                $ 887 "A_Touch_p[A_sel_v]=touch_xyz_get_middle(vr2_p1,vr2_p2,vr2_p3,vr2_p4)"
                A_Touch_p[A_sel_v]=touch_xyz_get_middle(vr2_p1,vr2_p2,vr2_p3,vr2_p4)
                $ 888 "var_4≔A_Touch_p[A_sel_v]"
                global var_4=A_Touch_p[A_sel_v]
                $ 889 "var_4≔pose_trans(var_4, p[a6_callar_vert/1000,0,0,0,0,0])"
                global var_4= pose_trans (var_4, p[a6_callar_vert/1000,0,0,0,0,0])
                $ 890 "var_5≔get_actual_tcp_pose()"
                global var_5= get_actual_tcp_pose ()
                $ 891 "var_5[2]=var_4[2]"
                var_5[2]=var_4[2]
                $ 892 "var_5≔pose_trans(var_5, p[0,0,0,0,d2r(10),0])"
                global var_5= pose_trans (var_5, p[0,0,0,0,d2r(10),0])
                $ 893 "MoveL"
                $ 894 "var_5" "breakAfter"
                movel(pose_trans(Base, var_5), a=0.1, v=0.1)
                $ 895 "vr2_p1_up≔contact_fun(p[0,0,0,0,0,0],[1,0,0],20000,20,20)"
                global vr2_p1_up=contact_fun(p[0,0,0,0,0,0],[1,0,0],20000,20,20)
                $ 896 "direction(p[0,0,0,0,0,0],[-1,0,0],20,120,160)"
                direction(p[0,0,0,0,0,0],[-1,0,0],20,120,160)
                $ 897 "direction(p[0,0,0,0,0,0],[0,1,0],10,120,160)"
                direction(p[0,0,0,0,0,0],[0,1,0],10,120,160)
                $ 898 "vr2_p2_up≔contact_fun(p[0,0,0,0,0,0],[1,0,0],20000,20,20)"
                global vr2_p2_up=contact_fun(p[0,0,0,0,0,0],[1,0,0],20000,20,20)
                $ 899 "direction(p[0,0,0,0,0,0],[-1,0,0],14,120,160)"
                direction(p[0,0,0,0,0,0],[-1,0,0],14,120,160)
                $ 900 "vr2_p3_up≔contact_fun(p[0,0,0,0,0,0],[0,1,0],20000,20,20)"
                global vr2_p3_up=contact_fun(p[0,0,0,0,0,0],[0,1,0],20000,20,20)
                $ 901 "direction(p[0,0,0,0,0,0],[0,-1,0],30,120,160)"
                direction(p[0,0,0,0,0,0],[0,-1,0],30,120,160)
                $ 902 "direction(p[0,0,0,0,0,0],[-1,0,0],20,120,160)"
                direction(p[0,0,0,0,0,0],[-1,0,0],20,120,160)
              end
              $ 903 "A_Touch_p[A_sel_v+9]=touch_4point(vr2_p1_up,vr2_p2_up,vr2_p3_up)"
              A_Touch_p[A_sel_v+9]=touch_4point(vr2_p1_up,vr2_p2_up,vr2_p3_up)
              $ 904 "A_Touch_p[A_sel_v+9]=ori_pose(A_Touch_p[A_sel_v+9],A_Touch_p[A_sel_v])"
              A_Touch_p[A_sel_v+9]=ori_pose(A_Touch_p[A_sel_v+9],A_Touch_p[A_sel_v])
            else:
              $ 905 "Else" "noBreak"
              $ 906 "If A_Touch_p[A_VR1]≟p[0,0,0,0,0,0]"
              if (A_Touch_p[A_VR1] == p[0,0,0,0,0,0]):
                $ 907 "Call MoveandTouchFun_3f"
                MoveandTouchFun_3f()
                $ 908 "touch_tmp≔A_Touch_p[A_sel_v]"
                global touch_tmp=A_Touch_p[A_sel_v]
                $ 909 "If A_Prepos_l[A_HOR_MR]≟p[0,0,0,0,0,0]"
                if (A_Prepos_l[A_HOR_MR] == p[0,0,0,0,0,0]):
                  $ 910 "direction(p[0,0,0,0,0,0],[0,1,0],8,120,160)"
                  direction(p[0,0,0,0,0,0],[0,1,0],8,120,160)
                  $ 911 "AAgcp≔get_actual_tcp_pose()"
                  global AAgcp= get_actual_tcp_pose ()
                  $ 912 "AAgangle≔up_right"
                  global AAgangle=p[.445203173045, -.406687378356, -.031125942276, 2.308490741423, -1.066468937023, 1.322151316133]
                  $ 913 "AAgtp≔p[AAgcp[0],AAgcp[1],AAgcp[2],AAgangle[3],AAgangle[4],AAgangle[5]]"
                  global AAgtp=p[AAgcp[0],AAgcp[1],AAgcp[2],AAgangle[3],AAgangle[4],AAgangle[5]]
                  $ 914 "MoveL"
                  $ 915 "AAgtp" "breakAfter"
                  movel(pose_trans(Base, AAgtp), a=0.08, v=0.08)
                end
                $ 917 "If b1_cell_info_R≠E and b1_cell_info_R≠e"
                if (b1_cell_info_R != E  and  b1_cell_info_R != e):
                  $ 918 "for_cal_zr≔contact_fun(p[0,0,0,0,0,0],[0,0,-1],20000,20,20)"
                  global for_cal_zr=contact_fun(p[0,0,0,0,0,0],[0,0,-1],20000,20,20)
                  $ 919 "touch_tmp[2]=for_cal_zr[2]"
                  touch_tmp[2]=for_cal_zr[2]
                end
                $ 920 "A_Touch_p[A_sel_v]=touch_tmp"
                A_Touch_p[A_sel_v]=touch_tmp
                $ 921 "for_cal_y_wel≔A_Touch_p[A_sel_v]"
                global for_cal_y_wel=A_Touch_p[A_sel_v]
                $ 922 "for_cal_x_wel≔A_Touch_p[A_sel_v]"
                global for_cal_x_wel=A_Touch_p[A_sel_v]
              else:
                $ 923 "Else" "noBreak"
                $ 924 "Call MoveFun"
                MoveFun()
                $ 925 "for_cal_y_wel≔contact_fun(p[0,0,0,0,0,0],[1,0,0],20000,20,20)"
                global for_cal_y_wel=contact_fun(p[0,0,0,0,0,0],[1,0,0],20000,20,20)
                $ 926 "direction(p[0,0,0,0,0,0],[-1,0,0],40,120,160)"
                direction(p[0,0,0,0,0,0],[-1,0,0],40,120,160)
                $ 927 "If A_Prepos_l[A_HOR_MR]≟p[0,0,0,0,0,0]"
                if (A_Prepos_l[A_HOR_MR] == p[0,0,0,0,0,0]):
                  $ 928 "direction(p[0,0,0,0,0,0],[0,-1,0],60,120,160)"
                  direction(p[0,0,0,0,0,0],[0,-1,0],60,120,160)
                  $ 929 "var_2≔contact_fun(p[0,0,0,0,0,0],[1,0,0],20000,20,20)"
                  global var_2=contact_fun(p[0,0,0,0,0,0],[1,0,0],20000,20,20)
                  $ 930 "direction(p[0,0,0,0,0,0],[-1,0,0],5,120,160)"
                  direction(p[0,0,0,0,0,0],[-1,0,0],5,120,160)
                  $ 931 "direction(p[0,0,0,0,0,0],[0,1,0],60,120,160)"
                  direction(p[0,0,0,0,0,0],[0,1,0],60,120,160)
                  $ 932 "direction(p[0,0,0,0,0,0],[1,0,0],10,120,160)"
                  direction(p[0,0,0,0,0,0],[1,0,0],10,120,160)
                  $ 933 "for_cal_x_wel≔contact_fun(p[0,0,0,0,0,0],[0,-1,0],20000,20,20)"
                  global for_cal_x_wel=contact_fun(p[0,0,0,0,0,0],[0,-1,0],20000,20,20)
                  $ 934 "direction(p[0,0,0,0,0,0],[0,1,0],20,120,160)"
                  direction(p[0,0,0,0,0,0],[0,1,0],20,120,160)
                  $ 935 "AAgcp≔get_actual_tcp_pose()"
                  global AAgcp= get_actual_tcp_pose ()
                  $ 936 "AAgangle≔up_right"
                  global AAgangle=p[.445203173045, -.406687378356, -.031125942276, 2.308490741423, -1.066468937023, 1.322151316133]
                  $ 937 "AAgtp≔p[AAgcp[0],AAgcp[1],AAgcp[2],AAgangle[3],AAgangle[4],AAgangle[5]]"
                  global AAgtp=p[AAgcp[0],AAgcp[1],AAgcp[2],AAgangle[3],AAgangle[4],AAgangle[5]]
                  $ 938 "MoveL"
                  $ 939 "AAgtp" "breakAfter"
                  movel(pose_trans(Base, AAgtp), a=0.1, v=0.1)
                  $ 941 "If b1_cell_info_R≠E and b1_cell_info_R≠e"
                  if (b1_cell_info_R != E  and  b1_cell_info_R != e):
                    $ 942 "for_cal_zr≔contact_fun(p[0,0,0,0,0,0],[0,0,-1],20000,20,20)"
                    global for_cal_zr=contact_fun(p[0,0,0,0,0,0],[0,0,-1],20000,20,20)
                    $ 943 "direction(p[0,0,0,0,0,0],[0,0,1],20,120,160)"
                    direction(p[0,0,0,0,0,0],[0,0,1],20,120,160)
                  end
                  $ 944 "direction(p[0,0,0,0,0,0],[-1,0,0],20,120,160)"
                  direction(p[0,0,0,0,0,0],[-1,0,0],20,120,160)
                end
                $ 945 "for_cal_rot≔A_Touch_p[A_VR1]"
                global for_cal_rot=A_Touch_p[A_VR1]
                $ 946 "If b1_cell_info_R≠E and b1_cell_info_R≠e"
                if (b1_cell_info_R != E  and  b1_cell_info_R != e):
                  $ 947 "A_Touch_p[A_sel_v]=p[for_cal_y_wel[0],for_cal_x_wel[1],for_cal_zr[2],for_cal_rot[3],for_cal_rot[4],for_cal_rot[5]]"
                  A_Touch_p[A_sel_v]=p[for_cal_y_wel[0],for_cal_x_wel[1],for_cal_zr[2],for_cal_rot[3],for_cal_rot[4],for_cal_rot[5]]
                  $ 948 "touch_tmp=p[for_cal_y_wel[0],for_cal_x_wel[1],for_cal_zr[2],for_cal_rot[3],for_cal_rot[4],for_cal_rot[5]]"
                  touch_tmp=p[for_cal_y_wel[0],for_cal_x_wel[1],for_cal_zr[2],for_cal_rot[3],for_cal_rot[4],for_cal_rot[5]]
                else:
                  $ 949 "Else" "noBreak"
                  $ 950 "A_Touch_p[A_sel_v]=p[for_cal_y_wel[0],for_cal_x_wel[1],for_cal_x_wel[2],for_cal_rot[3],for_cal_rot[4],for_cal_rot[5]]"
                  A_Touch_p[A_sel_v]=p[for_cal_y_wel[0],for_cal_x_wel[1],for_cal_x_wel[2],for_cal_rot[3],for_cal_rot[4],for_cal_rot[5]]
                  $ 951 "touch_tmp=p[for_cal_y_wel[0],for_cal_x_wel[1],for_cal_x_wel[2],for_cal_rot[3],for_cal_rot[4],for_cal_rot[5]]"
                  touch_tmp=p[for_cal_y_wel[0],for_cal_x_wel[1],for_cal_x_wel[2],for_cal_rot[3],for_cal_rot[4],for_cal_rot[5]]
                end
                $ 952 "If Scallup_check≟ False "
                if (Scallup_check ==   False  ):
                  $ 953 "touch_tmp≔pose_trans(touch_tmp,p[-(Touch_dis)/1000,0,0,0,0,0])"
                  global touch_tmp= pose_trans (touch_tmp,p[-(Touch_dis)/1000,0,0,0,0,0])
                  $ 954 "A_Touch_p[A_sel_v]=touch_tmp"
                  A_Touch_p[A_sel_v]=touch_tmp
                else:
                  $ 955 "Else" "noBreak"
                  $ 956 "Scallup_check≔ False "
                  global Scallup_check=  False
                end
                $ 957 "write_welder(4, False )"
                write_welder(4,  False  )
              end
            end
            $ 958 "b2_par_cd≔0"
            global b2_par_cd=0
            $ 959 "homeing()"
            homeing()
          else:
            $ 960 "Else" "noBreak"
            $ 961 "homeing()"
            homeing()
          end
          $ 962 "write_welder(4,False)"
          write_welder(4,False)
          $ 1019 "Touch After Offset"
          $ 1020 "touch_after_offset"
          $ 1021 "HOR"
          $ 1022 "If A_Prepos_l[A_HOR]≠p[0,0,0,0,0,0]"
          if (A_Prepos_l[A_HOR] != p[0,0,0,0,0,0]):
            $ 1023 "If b1_cell_info_L≟A or b1_cell_info_L≟C or b1_cell_info_L≟c"
            if (b1_cell_info_L == A  or  b1_cell_info_L == C  or  b1_cell_info_L == c):
              $ 1024 "If for_x_HOR≟p[0,0,0,0,0,0]"
              if (for_x_HOR == p[0,0,0,0,0,0]):
                $ 1025 "for_x_HOR≔A_Touch_p[A_VL1]"
                global for_x_HOR=A_Touch_p[A_VL1]
              end
              $ 1026 "If for_x_HOR≠p[0,0,0,0,0,0]"
              if (for_x_HOR != p[0,0,0,0,0,0]):
                $ 1027 "x_diff≔get_feature_pose(for_x_HOR,A_Touch_p[A_HOR])"
                global x_diff=get_feature_pose(for_x_HOR,A_Touch_p[A_HOR])
                $ 1028 "A_Touch_p[A_HOR]=pose_trans(A_Touch_p[A_HOR], p[x_diff[0],0,0,0,0,0])"
                A_Touch_p[A_HOR]= pose_trans (A_Touch_p[A_HOR], p[x_diff[0],0,0,0,0,0])
              end
            end
            $ 1029 "A_Touch_p[A_HOR]=pose_trans(A_Touch_p[A_HOR], p[offset_2f_begin/1000,0,0,0,0,0])"
            A_Touch_p[A_HOR]= pose_trans (A_Touch_p[A_HOR], p[offset_2f_begin/1000,0,0,0,0,0])
          end
          $ 1030 "VL1"
          $ 1031 "If A_Prepos_l[A_VL1]≠p[0,0,0,0,0,0]"
          if (A_Prepos_l[A_VL1] != p[0,0,0,0,0,0]):
            $ 1032 "If b1_cell_info_L≟A or b1_cell_info_L≟C or b1_cell_info_L≟c"
            if (b1_cell_info_L == A  or  b1_cell_info_L == C  or  b1_cell_info_L == c):
              $ 1033 "'3f only does not apply offset'"
              # '3f only does not apply offset'
              $ 1034 "If for_z_VL1≟p[0,0,0,0,0,0]"
              if (for_z_VL1 == p[0,0,0,0,0,0]):
                $ 1035 "for_z_VL1≔A_Touch_p[A_HOR]"
                global for_z_VL1=A_Touch_p[A_HOR]
              end
              $ 1036 "Comment"
              # Comment
              $ 1037 "If for_z_VL1≠p[0,0,0,0,0,0]"
              if (for_z_VL1 != p[0,0,0,0,0,0]):
                $ 1038 "z_diff≔get_feature_pose(for_z_VL1,A_Touch_p[A_VL1])"
                global z_diff=get_feature_pose(for_z_VL1,A_Touch_p[A_VL1])
                $ 1039 "A_Touch_p[A_VL1]=pose_trans(A_Touch_p[A_VL1], p[z_diff[0],0,0,0,0,0])"
                A_Touch_p[A_VL1]= pose_trans (A_Touch_p[A_VL1], p[z_diff[0],0,0,0,0,0])
              end
            end
            $ 1041 "A_Touch_p[A_VL1]=pose_trans(A_Touch_p[A_VL1], p[offset_3f_begin/1000,0,0,0,0,0])"
            A_Touch_p[A_VL1]= pose_trans (A_Touch_p[A_VL1], p[offset_3f_begin/1000,0,0,0,0,0])
          end
          $ 1042 "VL2"
          $ 1043 "If A_Prepos_l[A_VL2]≠p[0,0,0,0,0,0]"
          if (A_Prepos_l[A_VL2] != p[0,0,0,0,0,0]):
            $ 1044 "A_Touch_p[A_VL2]=pose_trans(A_Touch_p[A_VL2], p[offset_3f_begin/1000,0,0,0,0,0])"
            A_Touch_p[A_VL2]= pose_trans (A_Touch_p[A_VL2], p[offset_3f_begin/1000,0,0,0,0,0])
          end
          $ 1045 "HOR_R"
          $ 1046 "If A_Prepos_l[A_HOR_R]≠p[0,0,0,0,0,0]"
          if (A_Prepos_l[A_HOR_R] != p[0,0,0,0,0,0]):
            $ 1047 "If b1_cell_info_R≟A or b1_cell_info_R≟C or b1_cell_info_R≟c"
            if (b1_cell_info_R == A  or  b1_cell_info_R == C  or  b1_cell_info_R == c):
              $ 1048 "If for_x_HOR_R≟p[0,0,0,0,0,0]"
              if (for_x_HOR_R == p[0,0,0,0,0,0]):
                $ 1049 "for_x_HOR_R≔A_Touch_p[A_VR1]"
                global for_x_HOR_R=A_Touch_p[A_VR1]
              end
              $ 1050 "If for_x_HOR≠p[0,0,0,0,0,0]"
              if (for_x_HOR != p[0,0,0,0,0,0]):
                $ 1051 "x_diff≔get_feature_pose(for_x_HOR_R,A_Touch_p[A_HOR_R])"
                global x_diff=get_feature_pose(for_x_HOR_R,A_Touch_p[A_HOR_R])
                $ 1052 "A_Touch_p[A_HOR_R]=pose_trans(A_Touch_p[A_HOR_R], p[x_diff[0],0,0,0,0,0])"
                A_Touch_p[A_HOR_R]= pose_trans (A_Touch_p[A_HOR_R], p[x_diff[0],0,0,0,0,0])
              end
            end
            $ 1053 "A_Touch_p[A_HOR_R]=pose_trans(A_Touch_p[A_HOR_R], p[-offset_2f_begin/1000,0,0,0,0,0])"
            A_Touch_p[A_HOR_R]= pose_trans (A_Touch_p[A_HOR_R], p[-offset_2f_begin/1000,0,0,0,0,0])
          end
          $ 1054 "VR1"
          $ 1055 "If A_Prepos_l[A_VR1]≠p[0,0,0,0,0,0]"
          if (A_Prepos_l[A_VR1] != p[0,0,0,0,0,0]):
            $ 1056 "If b1_cell_info_R≟A or b1_cell_info_R≟C or b1_cell_info_R≟c"
            if (b1_cell_info_R == A  or  b1_cell_info_R == C  or  b1_cell_info_R == c):
              $ 1057 "If for_z_VR1≟p[0,0,0,0,0,0]"
              if (for_z_VR1 == p[0,0,0,0,0,0]):
                $ 1058 "for_z_VR1≔A_Touch_p[A_HOR_R]"
                global for_z_VR1=A_Touch_p[A_HOR_R]
              end
              $ 1059 "If for_z_VR1≠p[0,0,0,0,0,0]"
              if (for_z_VR1 != p[0,0,0,0,0,0]):
                $ 1060 "z_diff≔get_feature_pose(for_z_VR1,A_Touch_p[A_VR1])"
                global z_diff=get_feature_pose(for_z_VR1,A_Touch_p[A_VR1])
                $ 1061 "A_Touch_p[A_VR1]=pose_trans(A_Touch_p[A_VR1], p[z_diff[0],0,0,0,0,0])"
                A_Touch_p[A_VR1]= pose_trans (A_Touch_p[A_VR1], p[z_diff[0],0,0,0,0,0])
              end
            end
            $ 1063 "A_Touch_p[A_VR1]=pose_trans(A_Touch_p[A_VR1], p[offset_3f_begin/1000,0,0,0,0,0])"
            A_Touch_p[A_VR1]= pose_trans (A_Touch_p[A_VR1], p[offset_3f_begin/1000,0,0,0,0,0])
          end
          $ 1064 "VR2"
          $ 1065 "If A_Prepos_l[A_VR2]≠p[0,0,0,0,0,0]"
          if (A_Prepos_l[A_VR2] != p[0,0,0,0,0,0]):
            $ 1066 "A_Touch_p[A_VR2]=pose_trans(A_Touch_p[A_VR2], p[offset_3f_begin/1000,0,0,0,0,0])"
            A_Touch_p[A_VR2]= pose_trans (A_Touch_p[A_VR2], p[offset_3f_begin/1000,0,0,0,0,0])
          end
          $ 1067 "HOR_ML"
          $ 1068 "If A_Prepos_l[A_HOR_ML]≠p[0,0,0,0,0,0]"
          if (A_Prepos_l[A_HOR_ML] != p[0,0,0,0,0,0]):
            $ 1069 "A_Touch_p[A_HOR_M]=A_Touch_p[A_HOR_ML]"
            A_Touch_p[A_HOR_M]=A_Touch_p[A_HOR_ML]
            $ 1070 "x_welding_axis≔get_feature_pose(for_cal_x_wel,A_Touch_p[A_HOR_ML])"
            global x_welding_axis=get_feature_pose(for_cal_x_wel,A_Touch_p[A_HOR_ML])
            $ 1071 "A_Touch_p[A_HOR_M]=pose_trans(A_Touch_p[A_HOR_ML], p[x_welding_axis[0],0,0,0,0,0])"
            A_Touch_p[A_HOR_M]= pose_trans (A_Touch_p[A_HOR_ML], p[x_welding_axis[0],0,0,0,0,0])
            $ 1072 "A_Touch_p[A_HOR_M]=put_pose(A_Touch_p[A_HOR_M],0,for_cal_y_wel[0])"
            A_Touch_p[A_HOR_M]=put_pose(A_Touch_p[A_HOR_M],0,for_cal_y_wel[0])
            $ 1073 "A_Touch_p[A_HOR_M]=pose_trans(A_Touch_p[A_HOR_M], p[10/1000,0,0,0,0,0])"
            A_Touch_p[A_HOR_M]= pose_trans (A_Touch_p[A_HOR_M], p[10/1000,0,0,0,0,0])
            $ 1074 "If b1_cell_info_L≟C or b1_cell_info_L≟D"
            if (b1_cell_info_L == C  or  b1_cell_info_L == D):
              $ 1076 "x_welding_axis≔get_feature_pose(for_cal_x_wel,A_Touch_p[A_HOR_ML])"
              global x_welding_axis=get_feature_pose(for_cal_x_wel,A_Touch_p[A_HOR_ML])
              $ 1077 "A_Touch_p[A_HOR_ML]=pose_trans(A_Touch_p[A_HOR_ML],p[x_welding_axis[0],0,0,0,0,0])"
              A_Touch_p[A_HOR_ML]= pose_trans (A_Touch_p[A_HOR_ML],p[x_welding_axis[0],0,0,0,0,0])
              $ 1078 "A_Touch_p[A_HOR_ML]=pose_trans(A_Touch_p[A_HOR_ML],p[0/1000,0,0,0,0,0])"
              A_Touch_p[A_HOR_ML]= pose_trans (A_Touch_p[A_HOR_ML],p[0/1000,0,0,0,0,0])
            end
          end
          $ 1079 "HOR_MR"
          $ 1080 "If A_Prepos_l[A_HOR_MR]≠p[0,0,0,0,0,0]"
          if (A_Prepos_l[A_HOR_MR] != p[0,0,0,0,0,0]):
            $ 1082 "A_Touch_p[A_HOR_M]=A_Touch_p[A_HOR_MR]"
            A_Touch_p[A_HOR_M]=A_Touch_p[A_HOR_MR]
            $ 1083 "x_welding_axis≔get_feature_pose(for_cal_x_wel,A_Touch_p[A_HOR_MR])"
            global x_welding_axis=get_feature_pose(for_cal_x_wel,A_Touch_p[A_HOR_MR])
            $ 1084 "A_Touch_p[A_HOR_M]=pose_trans(A_Touch_p[A_HOR_M], p[x_welding_axis[0],0,0,0,0,0])"
            A_Touch_p[A_HOR_M]= pose_trans (A_Touch_p[A_HOR_M], p[x_welding_axis[0],0,0,0,0,0])
            $ 1085 "A_Touch_p[A_HOR_M]=put_pose(A_Touch_p[A_HOR_M],0,for_cal_y_wel[0])"
            A_Touch_p[A_HOR_M]=put_pose(A_Touch_p[A_HOR_M],0,for_cal_y_wel[0])
            $ 1086 "A_Touch_p[A_HOR_M]=pose_trans(A_Touch_p[A_HOR_M], p[-10/1000,0,0,0,0,0])"
            A_Touch_p[A_HOR_M]= pose_trans (A_Touch_p[A_HOR_M], p[-10/1000,0,0,0,0,0])
            $ 1087 "If b1_cell_info_R≟C or b1_cell_info_R≟D"
            if (b1_cell_info_R == C  or  b1_cell_info_R == D):
              $ 1089 "x_welding_axis≔get_feature_pose(for_cal_x_wel,A_Touch_p[A_HOR_MR])"
              global x_welding_axis=get_feature_pose(for_cal_x_wel,A_Touch_p[A_HOR_MR])
              $ 1090 "A_Touch_p[A_HOR_MR]=pose_trans(A_Touch_p[A_HOR_MR],p[x_welding_axis[0],0,0,0,0,0])"
              A_Touch_p[A_HOR_MR]= pose_trans (A_Touch_p[A_HOR_MR],p[x_welding_axis[0],0,0,0,0,0])
              $ 1091 "A_Touch_p[A_HOR_MR]=pose_trans(A_Touch_p[A_HOR_MR],p[-0/1000,0,0,0,0,0])"
              A_Touch_p[A_HOR_MR]= pose_trans (A_Touch_p[A_HOR_MR],p[-0/1000,0,0,0,0,0])
            end
          end
          $ 1092 "'Touch Remember On/OFF'"
          # 'Touch Remember On/OFF'
          $ 1093 "write_port_register(180,1)"
          write_port_register(180,1)
        else:
          $ 1094 "Else" "noBreak"
          $ 1095 "Ignore Touch and check error"
          $ 1096 "Auto_cur_cell≔0"
          global Auto_cur_cell=0
          $ 1097 "Loop Auto_cur_cell<Auto_total_cell"
          while (Auto_cur_cell<Auto_total_cell):
            $ 1098 "A_sel_v≔Auto_W_num[Auto_cur_cell]"
            global A_sel_v=Auto_W_num[Auto_cur_cell]
            $ 1099 "If A_sel_v<A_HOR_2path"
            if (A_sel_v<A_HOR_2path):
              $ 1100 "If A_Touch_p[A_sel_v]≟p[0,0,0,0,0,0]"
              if (A_Touch_p[A_sel_v] == p[0,0,0,0,0,0]):
                $ 1101 "write_port_register(142,120)"
                write_port_register(142,120)
                $ 1102 "Halt"
                halt
              end
            end
            $ 1103 "Auto_cur_cell≔Auto_cur_cell+1"
            global Auto_cur_cell=Auto_cur_cell+1
          end
          $ 1104 "Auto_cur_cell≔0"
          global Auto_cur_cell=0
        end
        $ 1105 "welding"
        $ 1106 "weldings"
        $ 1107 "Auto_cur_cell≔read_port_register(138)"
        global Auto_cur_cell= read_port_register (138)
        $ 1108 "time_cal_trig≔ True "
        global time_cal_trig=  True
        $ 1109 "Loop Auto_cur_cell<Auto_total_cell"
        while (Auto_cur_cell<Auto_total_cell):
          $ 1110 "write_port_register(138,Auto_cur_cell)"
          write_port_register(138,Auto_cur_cell)
          $ 1111 "running_trig≔ True "
          global running_trig=  True
          $ 1112 "'[2F_AB - 30] , [2F_CD_LEFT - 100] , [2F_CD_RIGHT - 150] , [3F - ELSE]'"
          # '[2F_AB - 30] , [2F_CD_LEFT - 100] , [2F_CD_RIGHT - 150] , [3F - ELSE]'
          $ 1113 "If Auto_W_num[Auto_cur_cell]≥100 and Auto_W_num[Auto_cur_cell]≤149"
          if (Auto_W_num[Auto_cur_cell] >= 100  and  Auto_W_num[Auto_cur_cell] <= 149):
            $ 1114 "'2F CD LEFT'"
            # '2F CD LEFT'
            $ 1115 "A_sel_v≔A_HOR"
            global A_sel_v=A_HOR
            $ 1116 "A_sel_v_end≔A_HOR_ML"
            global A_sel_v_end=A_HOR_ML
            $ 1117 "A_sel_v2≔A_HOR_M"
            global A_sel_v2=A_HOR_M
            $ 1118 "A_sel_v_end2≔A_HOR_R"
            global A_sel_v_end2=A_HOR_R
            $ 1119 "If floor(Auto_W_num[Auto_cur_cell]/10)≟10"
            if (floor(Auto_W_num[Auto_cur_cell]/10) == 10):
              $ 1120 "current_path≔1"
              global current_path=1
              $ 1121 "multi_path≔1"
              global multi_path=1
            else:
              $ 1122 "ElseIf floor(Auto_W_num[Auto_cur_cell]/10)≟11"
              if (floor(Auto_W_num[Auto_cur_cell]/10) == 11):
                $ 1123 "current_path≔2"
                global current_path=2
                $ 1124 "multi_path≔2"
                global multi_path=2
              else:
                $ 1125 "ElseIf floor(Auto_W_num[Auto_cur_cell]/10)≟12"
                if (floor(Auto_W_num[Auto_cur_cell]/10) == 12):
                  $ 1126 "current_path≔3"
                  global current_path=3
                  $ 1127 "multi_path≔3"
                  global multi_path=3
                else:
                  $ 1128 "ElseIf floor(Auto_W_num[Auto_cur_cell]/10)≟13"
                  if (floor(Auto_W_num[Auto_cur_cell]/10) == 13):
                    $ 1129 "current_path≔4"
                    global current_path=4
                    $ 1130 "multi_path≔4"
                    global multi_path=4
                  end
                end
              end
            end
            $ 1131 "current_2f≔current_2f+1"
            global current_2f=current_2f+1
            $ 1132 "CD_MLR≔ True "
            global CD_MLR=  True
            $ 1133 "write_port_register(135,A_HOR)"
            write_port_register(135,A_HOR)
            $ 1134 "write_port_register(136,current_2f)"
            write_port_register(136,current_2f)
            $ 1135 "If simulation_mode"
            if (simulation_mode):
              $ 1136 "Call welding_parameter_sim"
              welding_parameter_sim()
            else:
              $ 1137 "Else" "noBreak"
              $ 1138 "Call welding_parameter_init"
              welding_parameter_init()
            end
            $ 1139 "wv_direction≔1"
            global wv_direction=1
            $ 1140 "If Auto_W_num[Auto_cur_cell]%10≟4"
            if (Auto_W_num[Auto_cur_cell]%10 == 4):
              $ 1141 "A_sel_v≔A_HOR_R"
              global A_sel_v=A_HOR_R
              $ 1142 "Call MoveFun"
              MoveFun()
              $ 1143 "A_sel_v≔A_HOR"
              global A_sel_v=A_HOR
            else:
              $ 1144 "ElseIf Auto_W_num[Auto_cur_cell]%10≟0 or Auto_W_num[Auto_cur_cell]%10≟1 or Auto_W_num[Auto_cur_cell]%10≟2"
              if (Auto_W_num[Auto_cur_cell]%10 == 0  or  Auto_W_num[Auto_cur_cell]%10 == 1  or  Auto_W_num[Auto_cur_cell]%10 == 2):
                $ 1145 "Call MoveFun"
                MoveFun()
              end
            end
            $ 1146 "Call weav_welding_2f_CD"
            weav_welding_2f_CD()
          else:
            $ 1147 "ElseIf Auto_W_num[Auto_cur_cell]≥150 and Auto_W_num[Auto_cur_cell]≤189"
            if (Auto_W_num[Auto_cur_cell] >= 150  and  Auto_W_num[Auto_cur_cell] <= 189):
              $ 1148 "'2F CD RIGHT'"
              # '2F CD RIGHT'
              $ 1149 "A_sel_v≔A_HOR_R"
              global A_sel_v=A_HOR_R
              $ 1150 "A_sel_v_end≔A_HOR_MR"
              global A_sel_v_end=A_HOR_MR
              $ 1151 "A_sel_v2≔A_HOR_M"
              global A_sel_v2=A_HOR_M
              $ 1152 "A_sel_v_end2≔A_HOR"
              global A_sel_v_end2=A_HOR
              $ 1153 "If floor(Auto_W_num[Auto_cur_cell]/10)≟15"
              if (floor(Auto_W_num[Auto_cur_cell]/10) == 15):
                $ 1154 "current_path≔1"
                global current_path=1
                $ 1155 "multi_path≔1"
                global multi_path=1
              else:
                $ 1156 "ElseIf floor(Auto_W_num[Auto_cur_cell]/10)≟16"
                if (floor(Auto_W_num[Auto_cur_cell]/10) == 16):
                  $ 1157 "current_path≔2"
                  global current_path=2
                  $ 1158 "multi_path≔2"
                  global multi_path=2
                else:
                  $ 1159 "ElseIf floor(Auto_W_num[Auto_cur_cell]/10)≟17"
                  if (floor(Auto_W_num[Auto_cur_cell]/10) == 17):
                    $ 1160 "current_path≔3"
                    global current_path=3
                    $ 1161 "multi_path≔3"
                    global multi_path=3
                  else:
                    $ 1162 "ElseIf floor(Auto_W_num[Auto_cur_cell]/10)≟18"
                    if (floor(Auto_W_num[Auto_cur_cell]/10) == 18):
                      $ 1163 "current_path≔4"
                      global current_path=4
                      $ 1164 "multi_path≔4"
                      global multi_path=4
                    end
                  end
                end
              end
              $ 1165 "current_2f≔current_2f+1"
              global current_2f=current_2f+1
              $ 1166 "CD_MLR≔ False "
              global CD_MLR=  False
              $ 1167 "write_port_register(135,A_HOR)"
              write_port_register(135,A_HOR)
              $ 1168 "write_port_register(136,current_2f)"
              write_port_register(136,current_2f)
              $ 1169 "If simulation_mode"
              if (simulation_mode):
                $ 1170 "Call welding_parameter_sim"
                welding_parameter_sim()
              else:
                $ 1171 "Else" "noBreak"
                $ 1172 "Call welding_parameter_init"
                welding_parameter_init()
              end
              $ 1173 "wv_direction≔-1"
              global wv_direction=-1
              $ 1174 "If Auto_W_num[Auto_cur_cell]%10≟4"
              if (Auto_W_num[Auto_cur_cell]%10 == 4):
                $ 1175 "A_sel_v≔A_HOR"
                global A_sel_v=A_HOR
                $ 1176 "Call MoveFun"
                MoveFun()
                $ 1177 "A_sel_v≔A_HOR_R"
                global A_sel_v=A_HOR_R
              else:
                $ 1178 "ElseIf Auto_W_num[Auto_cur_cell]%10≟0 or Auto_W_num[Auto_cur_cell]%10≟1 or Auto_W_num[Auto_cur_cell]%10≟2"
                if (Auto_W_num[Auto_cur_cell]%10 == 0  or  Auto_W_num[Auto_cur_cell]%10 == 1  or  Auto_W_num[Auto_cur_cell]%10 == 2):
                  $ 1179 "Call MoveFun"
                  MoveFun()
                end
              end
              $ 1180 "Call weav_welding_2f_CD"
              weav_welding_2f_CD()
            else:
              $ 1181 "ElseIf Auto_W_num[Auto_cur_cell]≥30 and Auto_W_num[Auto_cur_cell]≤65"
              if (Auto_W_num[Auto_cur_cell] >= 30  and  Auto_W_num[Auto_cur_cell] <= 65):
                $ 1182 "'2F'"
                # '2F'
                $ 1183 "A_sel_v≔A_HOR"
                global A_sel_v=A_HOR
                $ 1184 "A_sel_v_end≔A_HOR_R"
                global A_sel_v_end=A_HOR_R
                $ 1185 "If floor(Auto_W_num[Auto_cur_cell]/10)≟3"
                if (floor(Auto_W_num[Auto_cur_cell]/10) == 3):
                  $ 1186 "current_path≔1"
                  global current_path=1
                  $ 1187 "multi_path≔1"
                  global multi_path=1
                else:
                  $ 1188 "ElseIf floor(Auto_W_num[Auto_cur_cell]/10)≟4"
                  if (floor(Auto_W_num[Auto_cur_cell]/10) == 4):
                    $ 1189 "current_path≔2"
                    global current_path=2
                    $ 1190 "multi_path≔2"
                    global multi_path=2
                  else:
                    $ 1191 "ElseIf floor(Auto_W_num[Auto_cur_cell]/10)≟5"
                    if (floor(Auto_W_num[Auto_cur_cell]/10) == 5):
                      $ 1192 "current_path≔3"
                      global current_path=3
                      $ 1193 "multi_path≔3"
                      global multi_path=3
                    else:
                      $ 1194 "ElseIf floor(Auto_W_num[Auto_cur_cell]/10)≟6"
                      if (floor(Auto_W_num[Auto_cur_cell]/10) == 6):
                        $ 1195 "current_path≔4"
                        global current_path=4
                        $ 1196 "multi_path≔4"
                        global multi_path=4
                      end
                    end
                  end
                end
                $ 1197 "current_2f≔current_2f+1"
                global current_2f=current_2f+1
                $ 1198 "write_port_register(135,A_HOR)"
                write_port_register(135,A_HOR)
                $ 1199 "write_port_register(136,current_2f)"
                write_port_register(136,current_2f)
                $ 1200 "If simulation_mode"
                if (simulation_mode):
                  $ 1201 "Call welding_parameter_sim"
                  welding_parameter_sim()
                else:
                  $ 1202 "Else" "noBreak"
                  $ 1203 "Call welding_parameter_init"
                  welding_parameter_init()
                end
                $ 1204 "If Auto_W_num[Auto_cur_cell]%10≟2"
                if (Auto_W_num[Auto_cur_cell]%10 == 2):
                  $ 1205 "A_sel_v≔A_HOR_R"
                  global A_sel_v=A_HOR_R
                  $ 1206 "Call MoveFun"
                  MoveFun()
                  $ 1207 "A_sel_v≔A_HOR"
                  global A_sel_v=A_HOR
                else:
                  $ 1208 "Else" "noBreak"
                  $ 1209 "Call MoveFun"
                  MoveFun()
                end
                $ 1210 "Call weav_welding_2f"
                weav_welding_2f()
              else:
                $ 1211 "Else" "noBreak"
                $ 1212 "A_sel_v≔Auto_W_num[Auto_cur_cell]"
                global A_sel_v=Auto_W_num[Auto_cur_cell]
                $ 1213 "write_port_register(135,A_sel_v)"
                write_port_register(135,A_sel_v)
                $ 1214 "current_path≔1"
                global current_path=1
                $ 1215 "current_2f≔0"
                global current_2f=0
                $ 1216 "write_port_register(136,current_2f)"
                write_port_register(136,current_2f)
                $ 1217 "If simulation_mode"
                if (simulation_mode):
                  $ 1218 "Call welding_parameter_sim"
                  welding_parameter_sim()
                else:
                  $ 1219 "Else" "noBreak"
                  $ 1220 "Call welding_parameter_init"
                  welding_parameter_init()
                end
                $ 1221 "A_sel_v_end≔A_sel_v+9"
                global A_sel_v_end=A_sel_v+9
                $ 1222 "Call weav_welding_3f"
                weav_welding_3f()
              end
            end
          end
          $ 1223 "Call reset_weld_param"
          reset_weld_param()
          $ 1226 "If get_move_trig≟1"
          if (get_move_trig == 1):
            $ 1227 "If get_next_number≠Auto_cur_cell"
            if (get_next_number != Auto_cur_cell):
              $ 1228 "Auto_cur_cell≔get_next_number"
              global Auto_cur_cell=get_next_number
            else:
              $ 1229 "Else" "noBreak"
              $ 1230 "Auto_cur_cell≔Auto_cur_cell+1"
              global Auto_cur_cell=Auto_cur_cell+1
            end
            $ 1231 "write_port_register(166,0)"
            write_port_register(166,0)
            $ 1232 "write_port_register(167,0)"
            write_port_register(167,0)
            $ 1233 "get_move_trig≔0"
            global get_move_trig=0
          else:
            $ 1234 "Else" "noBreak"
            $ 1235 "Auto_cur_cell≔Auto_cur_cell+1"
            global Auto_cur_cell=Auto_cur_cell+1
          end
        end
        $ 1236 "homeing()"
        homeing()
        $ 1237 "write_port_register(162,1)"
        write_port_register(162,1)
        $ 1238 "write_port_register(180,0)"
        write_port_register(180,0)
        thread_flag_301 = 1
      end
      if (a0_Job_Mode == 2):
        global thread_handler_301=run Thread_if_301()
        while (thread_flag_301 == 0):
          if not(a0_Job_Mode == 2):
            kill thread_handler_301
            thread_flag_301 = 2
          else:
            sync()
          end
        end
      else:
        thread_flag_301 = 2
      end
    end
    $ 1239 "Wait: 0.01"
    sleep(0.01)
    $ 1240 "after init auto"
    $ 1241 "If auto_on"
    if (auto_on):
      $ 1242 "write_port_register(202,0)"
      write_port_register(202,0)
      $ 1243 "timer_1: Stop"
      timer_1_is_counting = False
      $ 1244 "write_welder(0, False )"
      write_welder(0,  False  )
      $ 1245 "write_welder(4, False )"
      write_welder(4,  False  )
      $ 1246 "Call reset_weld_param"
      reset_weld_param()
      $ 1247 "multi_path≔1"
      global multi_path=1
      $ 1248 "auto_on≔ False "
      global auto_on=  False
      $ 1249 "current_2f≔0"
      global current_2f=0
      $ 1250 "get_center≔get_center_bak"
      global get_center=get_center_bak
      $ 1251 "vr2_p1≔p[0,0,0,0,0,0]"
      global vr2_p1=p[0,0,0,0,0,0]
      $ 1252 "welding_program≔ False "
      global welding_program=  False
      $ 1253 "start_num≔135"
      global start_num=135
      $ 1254 "Loop start_num<141"
      while (start_num<141):
        $ 1255 "write_port_register(start_num,0)"
        write_port_register(start_num,0)
        $ 1256 "start_num≔start_num+1"
        global start_num=start_num+1
      end
    end
  end
end
